FUNCTION_BLOCK FB_InternalPowerSupply
VAR CONSTANT
	//w_ID														: WORD := eObject_ID.InternalPowerSupply;
END_VAR

VAR
	IO: FB_InternalPowerSupply_IO;
	InternalPowerDemand: ST_PowerDemand;
	b_EMStopActive : BOOL := FALSE;
END_VAR

VAR_INPUT
	Set					:	ST_InternalPowerSupply_Set;
	BMSPowerstate		:	eHVDC_Powerstatus;
	b_ConditioningOnBatteryAllowed:	BOOL;
END_VAR

VAR_OUTPUT
	Get					:	ST_InternalPowerSupply_Get;
	b_HVDC_Enable		:	BOOL;
END_VAR

VAR
	ShutdownRequested	: BOOL := FALSE;	
	UPS					: FB_UPS;
END_VAR

(*
FB_InternalPowersupply
	Inputs:
		Power demand set by each applicable block, each with 3 booleans for 24V, 400VAc and HVDC:
			CoolingSystemPowerDemand	:	st_PowerDemand;
			PowerStackPowerDemand		:	st_PowerDemand;	
			UPSPowerDemand				:	st_PowerDemand;
			InternalPowerDemand			:	st_PowerDemand;
		
		Main system settings:	
			b_GeneralPowerEnable			: 	BOOL;	No power allowed without this being true. UPS only mode
		
		Input from powerstack. 400VAC available on busbar (via inverter or grid supply)	
			b_InternalBusbarACAvailable
		
		b_ShutdownUPS
			Kills UPS power, but only if other supplies are already down. 
	
	Outputs
		b_24VdcAvailable		
		b_HVDCAvailable			
		b_400VACAvailable		
			
		b_BMSForceOff 			//Output to FB_BMS to kill BMS supply voltage.
	
		UPS			//UPS data structure
	
		Events		
*)

//only if other power supplies are already down, UPS disable is allowed. Unwanted on live system.
IF (NOT (get.b_24VdcAvailable OR get.b_400VACAvailable OR get.b_HVDCAvailable)) AND set.b_ShutdownUPS THEN
	UPS.Shutdown();
END_IF

UPS(b_24v_available := get.b_24VdcAvailable, Get => get.UPS);
IO();
ACPowerControl();
DCPowerControl();
HVDCPowerControl();

METHOD PRIVATE ACPowerControl : BOOL
VAR
	AC_StartupDelay: TON := (PT := IPSParams.ACStartupDelay);
END_VAR
//AC control function
//Initial Diagnostics by reading fuse feedback
get.Events.b_GridInputFuseTripped 	:= NOT IO.GridFuseOK;
get.Events.b_CEEInputFuseTripped 	:= NOT IO.CeeFuseOK;

IF set.b_GeneralPowerEnable OR b_EMStopActive THEN
	//Grid power has priority over CEE plug
	IF 	IO.GridFuseOK AND set.b_InternalBusbarACAvailable THEN
		IO.SetACConnectionMode := 1;	//switch to grid AC
		AC_StartupDelay.IN := TRUE;	
	ELSIF IO.CEE_ACAvailable THEN 
		IO.SetACConnectionMode := 2;	//switch to CEE AC
		
		//not anymore
		//IF NOT Config.b_NeutralTransformer THEN //internal neutral transformer has longer startup time
		//	AC_StartupDelay.PT := IpsParams.ACStartupDelay+IPSParams.IntZPTStartupDelay;	
		//END_IF
		
		AC_StartupDelay.IN := TRUE;
	ELSE
		IO.SetACConnectionMode := 0;	//disable
		AC_StartupDelay.IN := FALSE;
	END_IF
ELSE 
	IO.SetACConnectionMode := 0;	//disable
	AC_StartupDelay.IN := FALSE;
END_IF

//after startup delay, internal 400VAC is available
get.b_400VACAvailable := AC_StartupDelay.Q;
END_METHOD

METHOD DCPowerControl : BOOL
VAR_INPUT
END_VAR
VAR
	DC_Required: BOOL;
	DCPSU_StartupDelay: TON := (PT := IPSParams.DCPSU_StartupDelay);
	ACPSU_StartupDelay: TON := (PT := IPSParams.ACPSU_StartupDelay);
END_VAR
ACPSU_StartupDelay.IN := get.b_400VACAvailable;
DCPSU_StartupDelay.IN := get.b_HVDCAvailable;

//if psu is not online after the startup delay, raise the fault status.
get.Events.b_ACPSUFault := ACPSU_StartupDelay.Q AND NOT IO.ACPSU_OK;
get.Events.b_DCPSUFault := DCPSU_StartupDelay.Q AND NOT IO.DCPSU_OK;

//if any of the psu's is online, 24V is available
get.b_24VdcAvailable := IO.ACPSU_OK OR IO.DCPSU_OK;

//All parts can demand 24V
DC_Required :=	set.CoolingSystemPowerDemand.b_Demand_24V OR 
				set.PowerStackPowerDemand.b_Demand_24V OR 
				set.UPSPowerDemand.b_Demand_24V;

//if no 400VAC available during 24VDC request, request HVDC ON for LVDC power				
internalPowerDemand.b_Demand_HVDC := DC_Required AND NOT get.b_400VACAvailable;
END_METHOD

METHOD PUBLIC EMstop : BOOL
VAR_INPUT
END_VAR
//return true if done
b_EMStopActive := TRUE;

//return true when all supplies are lost.
EMStop := not(get.b_24VdcAvailable OR get.b_400VACAvailable OR get.b_HVDCAvailable);
END_METHOD

METHOD GetDiagnostics 
VAR_IN_OUT
	AddError		: ARRAY [*] OF FB_AddErrorST;
	a_ActiveEvents	: ARRAY [*] OF ST_ErrorStruct;
	w_Index			: WORD;
END_VAR

VAR_OUTPUT
	b_errorActive	: BOOL;
	b_warningActive	: BOOL;
END_VAR

VAR
	by_errCt	: BYTE;
	by_warnCt	: BYTE;
	w_ID		: WORD;
END_VAR

//check if this call works:
UPS.GetDiagnostics(AddError := AddError, a_ActiveEvents := a_ActiveEvents, w_Index := w_Index, b_errorActive => b_errorActive, b_warningActive => b_warningActive);

(*IPS*)
	(*AC PSU fault*)		AddError[w_Index](
			in_b_ErrorTrig			:= Get.Events.b_ACPSUFault,
			out_ST_Error			:= a_ActiveEvents[w_Index],
			w_ID					:= 1 + w_ID,
			s_Message				:= 'AC PSU fault',
			e_sev					:= eSeverity.Warning,
			);
		IF AddError[w_Index].b_out THEN by_WarnCt := by_WarnCt + 1; END_IF;
		w_Index := w_Index +1;
		
	(*DC PSU fault*)		AddError[w_Index](
			in_b_ErrorTrig			:= Get.Events.b_DCPSUFault,
			out_ST_Error			:= a_ActiveEvents[w_Index],
			w_ID					:= 1 + w_ID,
			s_Message				:= 'DC PSU fault',
			e_sev					:= eSeverity.Warning,
			);
		IF AddError[w_Index].b_out THEN by_WarnCt := by_WarnCt + 1; END_IF;
		w_Index := w_Index +1;
	
	(*24V fault*)		AddError[w_Index](
			in_b_ErrorTrig			:= Get.Events.b_DCPSUFault AND Get.Events.b_ACPSUFault,
			out_ST_Error			:= a_ActiveEvents[w_Index],
			w_ID					:= 1 + w_ID,
			s_Message				:= '24V supply failed',
			e_sev					:= eSeverity.QuickShutdown,
			);
		IF AddError[w_Index].b_out THEN by_errCt := by_errCt + 1; END_IF;
		w_Index := w_Index +1;	
		
	(*CEE fuse tripped*)		AddError[w_Index](
			in_b_ErrorTrig			:= Get.Events.b_CEEInputFuseTripped,
			out_ST_Error			:= a_ActiveEvents[w_Index],
			w_ID					:= 1 + w_ID,
			s_Message				:= 'CEE Standby power input fuse error',
			e_sev					:= eSeverity.Warning,
			in_b_AutoClear			:= TRUE,
			
			);
		IF AddError[w_Index].b_out THEN by_WarnCt := by_WarnCt + 1; END_IF;
		w_Index := w_Index +1;
	
	(*internal grid fuse fault*)		AddError[w_Index](
			in_b_ErrorTrig		:= Get.Events.b_GridInputFuseTripped,
			out_ST_Error			:= a_ActiveEvents[w_Index],
			w_ID					:= 1 + w_ID,
			s_Message				:= 'Internal supply Grid fuse error',
			e_sev					:= eSeverity.QuickShutdown,
			in_b_AutoClear			:= TRUE,
			);
		IF AddError[w_Index].b_out THEN by_errCt := by_errCt + 1; END_IF;
		w_Index := w_Index +1;
		
	(*EMSTOP HVDC shutdown failed*)		AddError[w_Index](
			in_b_ErrorTrig			:= Get.Events.b_HVDCShutdownTimeExceeded,
			out_ST_Error			:= a_ActiveEvents[w_Index],
			w_ID					:= 1 + w_ID,
			s_Message				:= 'HVDC shutdown sequence failed',
			e_sev					:= eSeverity.QuickShutdown,			//<-- already in emstop, but this is a severe error
			);
		IF AddError[w_Index].b_out THEN by_errCt := by_errCt + 1; END_IF;
		w_Index := w_Index +1;
END_METHOD

METHOD PRIVATE HVDCPowerControl : BOOL
VAR_INPUT
END_VAR

//The powerstack demands HVDC directly. 
IF b_EMStopActive THEN
	b_HVDC_Enable := FALSE;
ELSE
	b_HVDC_Enable := set.PowerStackPowerDemand.b_Demand_HVDC 
		OR (InternalPowerDemand.b_Demand_HVDC AND b_ConditioningOnBatteryAllowed AND NOT ShutdownRequested);
END_IF						

IF BMSPowerState = eHVDC_Powerstatus.ON THEN
	get.b_HVDCAvailable := TRUE;
ELSE
	get.b_HVDCAvailable := FALSE;
END_IF
END_METHOD

METHOD Reset : BOOL
VAR_INPUT
END_VAR
//reset system
//return true if ok

b_EMStopActive 					:= 	FALSE;
IO.b_InternalHVDCConnected		:=	TRUE;

Reset := NOT get.Events.b_GridInputFuseTripped;
END_METHOD

METHOD SystemShutdown : BOOL
VAR_INPUT
	b_force		:	Bool;
END_VAR

IF B_force THEN
	IO.SetACConnectionMode 		:= 	0;
	IO.b_InternalHVDCConnected	:=	FALSE;
	IO.Write();

	UPS.Shutdown();
ELSE
	//no unforced shutdown allowed if HVDC is still online.
	//if HVDC offline, disable AC inputs and decouple HV contactors
	//Wait for 400VAC and 24V to be offline, then kill the UPS
	IF NOT get.b_HVDCAvailable THEN
		IO.b_InternalHVDCConnected := 0;
		IO.SetACConnectionMode 		:= 	0;
		IF NOT get.b_400VACAvailable AND get.b_24VdcAvailable THEN
			UPS.Shutdown();
		END_IF
	END_IF
END_IF
END_METHOD

END_FUNCTION_BLOCK

(* stored: Version 1.1.0.1, ProductVersion 3.1.4024.12
   POU FB_InternalPowerSupply: Id {99b5595d-91f9-4503-8fb7-aed8af10f6d8}, SpecialFunc None
   Method ACPowerControl: Id {5916b7c6-c369-43a6-ad0f-f820d571c778}
   Method DCPowerControl: Id {4cfaa935-ee98-4c42-8d5b-fbc6199322b8}
   Method EMstop: Id {4866248a-59ca-4029-a026-7364cef193b4}
   Method GetDiagnostics: Id {f562ae03-1873-4d82-904d-4e0cc41d7903}
   Method HVDCPowerControl: Id {ed7ee3c2-5980-4244-9ba9-7c622b5d790a}
   Method Reset: Id {d1725ace-f077-4c1f-9e1a-d4d8e986182f}
   Method SystemShutdown: Id {3b87d144-400f-4b3a-bef6-5aea1582308c} *)
